(* IEC 61131-3 sources: Internship/XML, 2 files *)

(* ---- Sim2Twin_controlsystem_pos_Discrete.st ---- *)
(*
 *
 * File: Sim2Twin_controlsystem_pos_Discrete.st
 *
 * IEC 61131-3 Structured Text (ST) code generated for subsystem "Sim2Twin_controlsystem_pos_Discrete/FB_ControlBlockWithMonitoring"
 *
 * Model name                      : Sim2Twin_controlsystem_pos_Discrete
 * Model version                   : 1.15
 * Model creator                   : Emila
 * Model last modified by          : Green Crane Testbed
 * Model last modified on          : Fri Nov 08 12:08:07 2024
 * Model sample time               : 0.001s
 * Subsystem name                  : Sim2Twin_controlsystem_pos_Discrete/FB_ControlBlockWithMonitoring
 * Subsystem sample time           : 0.001s
 * Simulink PLC Coder version      : 24.2 (R2024b) 21-Jun-2024
 * ST code generated on            : Fri Nov 08 12:25:28 2024
 *
 * Target IDE selection            : Beckhoff TwinCAT 3
 * Test Bench included             : No
 *
 *)
FUNCTION_BLOCK c_FB_ControlBlockWithMonito
VAR_INPUT
    ssMethodType: SINT;
    X_real: LREAL;
    X: LREAL;
    X_dot: LREAL;
    bEnableU: BOOL;
    bEnablePID: BOOL;
    Kp: LREAL;
    Ki: LREAL;
    Kd: LREAL;
    Ps: LREAL;
    Pa: LREAL;
    Pb: LREAL;
    u_filtered: LREAL;
END_VAR
VAR_OUTPUT
    U: LREAL;
    PID_OUT: LREAL;
    Error: LREAL;
    u_Unfiltered: LREAL;
END_VAR
VAR
    c_DiscreteTimeIntegrator_DS: LREAL;
    DiscreteTransferFcn_states: LREAL;
    UD_DSTATE: LREAL;
END_VAR
VAR_TEMP
    rtb_TSamp: LREAL;
    temp1: LREAL;
    temp2: LREAL;
END_VAR
CASE ssMethodType OF
    SS_INITIALIZE:
        (* SystemInitialize for Atomic SubSystem: '<Root>/FB_ControlBlockWithMonitoring' *)
        (* InitializeConditions for DiscreteTransferFcn: '<S2>/Discrete Transfer Fcn' *)
        DiscreteTransferFcn_states := 0.0;
        (* InitializeConditions for DiscreteIntegrator: '<S2>/Discrete-Time Integrator' *)
        c_DiscreteTimeIntegrator_DS := 0.0;
        (* InitializeConditions for UnitDelay: '<S4>/UD'
         *
         * Block description for '<S4>/UD':
         *
         *  Store in Global RAM *)
        UD_DSTATE := 0.0;
        (* End of SystemInitialize for SubSystem: '<Root>/FB_ControlBlockWithMonitoring' *)
    SS_STEP:
        (* Outputs for Atomic SubSystem: '<Root>/FB_ControlBlockWithMonitoring' *)
        (* Sum: '<S1>/Sum1' incorporates:
         *  Outport: '<Root>/Error' *)
        Error := X - X_real;
        (* SampleTimeMath: '<S4>/TSamp' incorporates:
         *  DiscreteTransferFcn: '<S2>/Discrete Transfer Fcn'
         *
         * About '<S4>/TSamp':
         *  y = u * K where K = 1 / ( w * Ts )
         *   *)
        rtb_TSamp := (0.0009995 * DiscreteTransferFcn_states) * 1000.0;
        (* Switch: '<S1>/Switch' incorporates:
         *  Constant: '<S1>/Constant'
         *  DiscreteIntegrator: '<S2>/Discrete-Time Integrator'
         *  Outport: '<Root>/Error'
         *  Product: '<S2>/Product'
         *  Product: '<S2>/Product1'
         *  Product: '<S2>/Product2'
         *  Sum: '<S2>/Sum1'
         *  Sum: '<S4>/Diff'
         *  UnitDelay: '<S4>/UD'
         *
         * Block description for '<S4>/Diff':
         *
         *  Add in CPU
         *
         * Block description for '<S4>/UD':
         *
         *  Store in Global RAM *)
        IF bEnablePID THEN
            U := ((Kp * Error) + (Ki * c_DiscreteTimeIntegrator_DS)) + ((rtb_TSamp - UD_DSTATE) * Kd);
        ELSE
            U := 0.0;
        END_IF;
        (* End of Switch: '<S1>/Switch' *)

        (* Saturate: '<S1>/Saturation1' *)
        IF U > 1.0 THEN
            PID_OUT := 1.0;
        ELSIF U >= -1.0 THEN
            PID_OUT := U;
        ELSE
            PID_OUT := -1.0;
        END_IF;
        (* End of Saturate: '<S1>/Saturation1' *)

        (* Switch: '<S1>/Switch1' incorporates:
         *  Constant: '<S1>/Constant1'
         *  Sum: '<S1>/Sum' *)
        IF bEnableU THEN
            U := u_filtered + PID_OUT;
        ELSE
            U := 0.0;
        END_IF;
        (* End of Switch: '<S1>/Switch1' *)

        (* Saturate: '<S1>/Saturation' *)
        IF U > 1.0 THEN
            (* Outport: '<Root>/U' *)
            U := 1.0;
        ELSIF U < -1.0 THEN
            (* Outport: '<Root>/U' *)
            U := -1.0;
        END_IF;
        (* End of Saturate: '<S1>/Saturation' *)

        (* MATLAB Function: '<S1>/V2Q2u' *)
        (* MATLAB Function 'FB_ControlBlockWithMonitoring/V2Q2u': '<S3>:1' *)
        (* '<S3>:1:3' phi = 0.7130; *)
        (* '<S3>:1:4' A = 33.1/100^2; *)
        (* Area *)
        (* '<S3>:1:5' BW = 0; *)
        (* deadband *)
        (* '<S3>:1:6' SpoolTravel = 7; *)
        (* Maximum Spool Travel *)
        (* '<S3>:1:7' a = (SpoolTravel-BW)/25; *)
        (* Valve Slope Characteristic [mm/(L/min)] *)
        (* '<S3>:1:8' dP_0 = 7e5; *)
        (* Pressure drop with compansator *)
        (* '<S3>:1:10' if x_dot > 0 *)
        IF X_dot > 0.0 THEN
            (* '<S3>:1:11' Q = x_dot * A; *)
            (* Wanted Flow *)
            (* '<S3>:1:12' dP = (Ps-Pa)*1e5; *)
            (* '<S3>:1:13' dp_ref = abs(dP_0/dP); *)
            (* dp_ref = 1; *)
            (* '<S3>:1:15' Q_star = (Q * sqrt(dp_ref)) * 6e4; *)
            (* Referance Flow [L/min] *)
            (* '<S3>:1:16' u = (Q_star * a + BW)/SpoolTravel; *)
            temp2 := ABS(700000.0 / ((Ps - Pa) * 100000.0));
            u_Unfiltered := (((SQRT(temp2) * (X_dot * 0.00331)) * 60000.0) * 0.28) / 7.0;
            (* Control Signal [-1, 1] *)
        ELSIF X_dot < 0.0 THEN
            (* '<S3>:1:18' elseif x_dot < 0 *)
            (* '<S3>:1:19' Q = x_dot * (A*phi); *)
            (* Wanted Flow *)
            (* '<S3>:1:20' dP = (Ps-Pb)*1e5; *)
            (* '<S3>:1:21' dp_ref = abs(dP_0/dP); *)
            (* dp_ref = 1; *)
            (* '<S3>:1:23' Q_star = (Q * sqrt(dp_ref)) * 6e4; *)
            (* Referance Flow [L/min] *)
            (* '<S3>:1:24' u = (Q_star * a - BW)/SpoolTravel; *)
            temp1 := ABS(700000.0 / ((Ps - Pb) * 100000.0));
            u_Unfiltered := (((SQRT(temp1) * (X_dot * 0.00236003)) * 60000.0) * 0.28) / 7.0;
            (* Control Signal [-1, 1] *)
        ELSE
            (* '<S3>:1:26' else *)
            (* '<S3>:1:27' u = 0; *)
            u_Unfiltered := 0.0;
        END_IF;
        (* End of MATLAB Function: '<S1>/V2Q2u' *)

        (* Saturate: '<S1>/Saturation2' *)
        IF u_Unfiltered > 1.0 THEN
            (* Outport: '<Root>/u_Unfiltered' *)
            u_Unfiltered := 1.0;
        ELSIF u_Unfiltered < -1.0 THEN
            (* Outport: '<Root>/u_Unfiltered' *)
            u_Unfiltered := -1.0;
        END_IF;
        (* End of Saturate: '<S1>/Saturation2' *)

        (* Update for DiscreteTransferFcn: '<S2>/Discrete Transfer Fcn' incorporates:
         *  Outport: '<Root>/Error' *)
        DiscreteTransferFcn_states := Error - (-0.999 * DiscreteTransferFcn_states);
        (* Update for DiscreteIntegrator: '<S2>/Discrete-Time Integrator' incorporates:
         *  Outport: '<Root>/Error' *)
        c_DiscreteTimeIntegrator_DS := (0.001 * Error) + c_DiscreteTimeIntegrator_DS;
        (* Update for UnitDelay: '<S4>/UD'
         *
         * Block description for '<S4>/UD':
         *
         *  Store in Global RAM *)
        UD_DSTATE := rtb_TSamp;
        (* End of Outputs for SubSystem: '<Root>/FB_ControlBlockWithMonitoring' *)
END_CASE;
END_FUNCTION_BLOCK
VAR_GLOBAL CONSTANT
    SS_INITIALIZE: SINT := 0;
    SS_STEP: SINT := 1;
END_VAR

(* ---- Sim2Twin_controlsystem_spd_Discrete.st ---- *)
(*
 *
 * File: Sim2Twin_controlsystem_spd_Discrete.st
 *
 * IEC 61131-3 Structured Text (ST) code generated for subsystem "Sim2Twin_controlsystem_spd_Discrete/FB_Joystick"
 *
 * Model name                      : Sim2Twin_controlsystem_spd_Discrete
 * Model version                   : 1.7
 * Model creator                   : Emila
 * Model last modified by          : Green Crane Testbed
 * Model last modified on          : Mon Nov 04 13:47:16 2024
 * Model sample time               : 0.001s
 * Subsystem name                  : Sim2Twin_controlsystem_spd_Discrete/FB_Joystick
 * Subsystem sample time           : 0.001s
 * Simulink PLC Coder version      : 24.2 (R2024b) 21-Jun-2024
 * ST code generated on            : Mon Nov 04 14:46:34 2024
 *
 * Target IDE selection            : Beckhoff TwinCAT 3
 * Test Bench included             : No
 *
 *)
FUNCTION_BLOCK FB_Joystick
VAR_INPUT
    ssMethodType: SINT;
    Joystick: LREAL;
    XRealRef: LREAL;
END_VAR
VAR_OUTPUT
    fPositionReferance_m: LREAL;
    fVelocityReferance_ms: LREAL;
END_VAR
VAR
    c_DiscreteTimeIntegrator_IC: USINT;
    c_DiscreteTimeIntegrator_DS: LREAL;
END_VAR
CASE ssMethodType OF
    SS_INITIALIZE:
        (* SystemInitialize for Atomic SubSystem: '<Root>/FB_Joystick' *)
        (* InitializeConditions for DiscreteIntegrator: '<S1>/Discrete-Time Integrator' *)
        c_DiscreteTimeIntegrator_IC := 1;
        (* End of SystemInitialize for SubSystem: '<Root>/FB_Joystick' *)
    SS_STEP:
        (* Outputs for Atomic SubSystem: '<Root>/FB_Joystick' *)
        (* Gain: '<S1>/Gain' *)
        fVelocityReferance_ms := 0.1 * Joystick;
        (* DiscreteIntegrator: '<S1>/Discrete-Time Integrator' *)
        IF c_DiscreteTimeIntegrator_IC <> 0 THEN
            c_DiscreteTimeIntegrator_DS := XRealRef;
            IF c_DiscreteTimeIntegrator_DS > 0.45 THEN
                c_DiscreteTimeIntegrator_DS := 0.45;
            ELSIF c_DiscreteTimeIntegrator_DS < 0.0 THEN
                c_DiscreteTimeIntegrator_DS := 0.0;
            END_IF;
        END_IF;
        (* Outport: '<Root>/fPositionReferance_m' incorporates:
         *  DiscreteIntegrator: '<S1>/Discrete-Time Integrator' *)
        fPositionReferance_m := c_DiscreteTimeIntegrator_DS;
        (* Update for DiscreteIntegrator: '<S1>/Discrete-Time Integrator' *)
        c_DiscreteTimeIntegrator_IC := 0;
        c_DiscreteTimeIntegrator_DS := (0.001 * fVelocityReferance_ms) + c_DiscreteTimeIntegrator_DS;
        IF c_DiscreteTimeIntegrator_DS > 0.45 THEN
            c_DiscreteTimeIntegrator_DS := 0.45;
        ELSIF c_DiscreteTimeIntegrator_DS < 0.0 THEN
            c_DiscreteTimeIntegrator_DS := 0.0;
        END_IF;
        (* End of Update for DiscreteIntegrator: '<S1>/Discrete-Time Integrator' *)
        (* End of Outputs for SubSystem: '<Root>/FB_Joystick' *)
END_CASE;
END_FUNCTION_BLOCK
VAR_GLOBAL CONSTANT
    SS_INITIALIZE: SINT := 0;
    SS_STEP: SINT := 1;
END_VAR
